DATA_BLOCK "Station5LoadData"
{ S7_Optimized_Access := 'FALSE' }
VERSION : 0.1
NON_RETAIN
// ATTRIBUTES
// AUTO_NUMBER = False
// BLOCK_NUMBER = 518
// END_ATTRIBUTES
   STRUCT
      "PLC.PartTypeID" : Int;
      "PLC.Station5RecipeNo" : Int;
      "PLC.Station5DMXCode" : String[128];
      "PLC.SubPartSN1" : String[128];
      "MES.ErrorCode" : Int;
      "MES.StatusBits" : DInt;
      "MES.Cycle_ID" : DInt;
      "MES.Unit_ParttypeID" : Int;
   END_STRUCT;


BEGIN

END_DATA_BLOCK

